FUNCTION_BLOCK Hiss
  (* Version 0.1, 2005-05-13, MF  BL, Chalmers *)
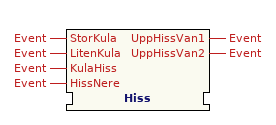
  EVENT_INPUT
    StorKula;
    LitenKula;
    KulaHiss;
    HissNere;
  END_EVENT
  EVENT_OUTPUT
    UppHissVan1;
    UppHissVan2;
  END_EVENT
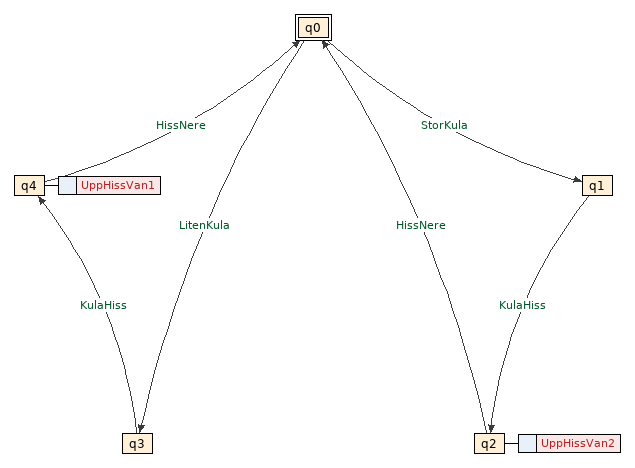
  EC_STATES
    q0;
    q1;
    q2 : -> UppHissVan2;
    q3;
    q4 : -> UppHissVan1;
  END_STATES
  EC_TRANSITIONS
    q0 TO q1 := StorKula;
    q1 TO q2 := KulaHiss;
    q0 TO q3 := LitenKula;
    q3 TO q4 := KulaHiss;
    q2 TO q0 := HissNere;
    q4 TO q0 := HissNere;
  END_TRANSITIONS
END_FUNCTION_BLOCK
